(* IEC 61131-3 sources: codesys-mcp-toolkit/standalone-sync/sources_st/511_05/Util, 8 files *)

(* ---- E_InfluxType.dut.st ---- *)
// @OBJECT_ID: 731e7745-b82f-47eb-ba89-92034cdd1c59
// @DECLARATION
TYPE E_InfluxType :
(
    REAL_TYPE,
    INT_TYPE,
    BOOL_TYPE
);
END_TYPE

(* ---- E_InfluxType_1.dut.st ---- *)
// @OBJECT_ID: 96c42348-4289-44bb-9086-91ce752858fa
// @DECLARATION
TYPE E_InfluxType_1 :
(
    REAL_TYPE,
    INT_TYPE,
    BOOL_TYPE
);
END_TYPE

(* ---- U_WordToReal.dut.st ---- *)
// @OBJECT_ID: 3d2ce4b8-1645-47ac-8a08-67d49366f794
// @DECLARATION
TYPE U_WordToReal :
UNION
    dwValue : DWORD; // Используется для битовых операций
    rValue  : REAL;  // Используется для получения результата
END_UNION
END_TYPE

(* ---- AIToFloat.func.st ---- *)
// @OBJECT_ID: 807a566b-cc68-4261-8820-1605cd0b0d30
// @DECLARATION
	FUNCTION AIToFloat : REAL
VAR_INPUT
	In:UINT;
	Lo,Hi:REAL;
END_VAR
VAR
END_VAR

// @IMPLEMENTATION
AIToFloat:=(UINT_TO_REAL(In)-10000.0)/40000.0*Hi+Lo;
//AIToFloat:=(UINT_TO_REAL(In)-0.0)/50000.0*Hi+Lo;

(* ---- FC_ModbusToRealSwapped.func.st ---- *)
// @OBJECT_ID: 0315c496-40b5-48b0-ae72-f392c63e890a
// @DECLARATION
FUNCTION FC_ModbusToRealSwapped : REAL
VAR_INPUT
    wWord1   : WORD;   (* Первое слово из Modbus (например, 53126) *)
    wWord2   : WORD;   (* Второе слово из Modbus (например, 0) *)
END_VAR
VAR
    dwTarget : DWORD;  (* Буфер для сборки 32-битного значения *)
    wTemp1   : WORD;   (* Временные переменные для перестановки байт *)
    wTemp2   : WORD;
    pReal    : POINTER TO REAL; (* Указатель для копирования памяти *)
END_VAR

// @IMPLEMENTATION

(* 1. Переставляем байты внутри каждого слова *)
wTemp1 := ROR(wWord1, 8); (* 0xED0C станет 0x0CED *)
wTemp2 := ROR(wWord2, 8); (* 0x0000 останется 0x0000 *)

(* 2. Собираем DWORD в режиме Little-Endian (wTemp2 сдвигаем в старшие биты) *)
dwTarget := SHL(WORD_TO_DWORD(wTemp2), 16) OR WORD_TO_DWORD(wTemp1);
(* На выходе соберется строка 0x41CD0000 *)

(* 3. Копируем область памяти в REAL *)
pReal := ADR(dwTarget);
FC_ModbusToRealSwapped := pReal^;

(* ---- FloatToAI.func.st ---- *)
// @OBJECT_ID: 9798738f-911b-4eef-bb17-69dfaa9c6f1e
// @DECLARATION
FUNCTION FloatToAI : UINT
VAR_INPUT
	In:REAL;

END_VAR
VAR
END_VAR

// @IMPLEMENTATION
FloatToAI:=REAL_TO_UINT(In/100.0*40000.0+10000.0);

(* ---- Check_Block.fb.st ---- *)
// @OBJECT_ID: a53145cf-05f5-44e2-98c8-5640a1ec8c65
// @DECLARATION
FUNCTION_BLOCK Check_Block
VAR_INPUT
	State_Mixer : BOOL;
	Weight : REAL;
END_VAR
VAR_OUTPUT
	State_Block : BOOL;
	State_Block_P102 : BOOL;
END_VAR
VAR
END_VAR

// @IMPLEMENTATION
IF NOT State_Mixer THEN
	State_Block := TRUE;
ELSE
	State_Block := FALSE;
END_IF;
IF Weight > 3000 THEN
	State_Block_P102 := TRUE;
ELSE
	State_Block_P102 := FALSE;
END_IF;

(* ---- FB_InfluxUdpSender.fb.st ---- *)
// @OBJECT_ID: e559a9a1-9e90-4a38-bf45-4143c502a1fc
// @DECLARATION
FUNCTION_BLOCK FB_InfluxUdpSender
VAR_INPUT
	sSendData : STRING(2000); // Data to send
    sIPInflux : STRING :='192.168.215.5'; // InfluxIP
    uiPortInflux : UINT := 8089; // Influx port
END_VAR
VAR
	eState: 			CLIENT_STATE;								// Шаг состояния клиента

	fbUdpPeer: 			NBS.UDP_Peer;								// ФБ создания UDP-пира
	fbUdpSend: 			NBS.UDP_Send;								// ФБ отправки данных
	sendData : STRING(2000); // Data to send
    numberOfBytesToSend : UDINT := 0; // Number of bytes to send
	influxIP: NBS.IP_ADDR;

	fbSendTrig:			R_TRIG;										// Триггер записи

	blinker:BLINK;
	TimeCycle: TIME:= T#10S;
	bStart : BOOL := FALSE;
END_VAR

// @IMPLEMENTATION
	blinker(ENABLE:=bStart,timelow:=TimeCycle, timehigh:=T#1S);

CASE eState OF

	CLIENT_STATE.CREATE:	// создаем UDP-пира на заданном порту

		fbUdpPeer
		(
			xEnable		:= TRUE,
			ipAddr		:= ,
			uiPort		:= ,
			ipMultiCast	:= ,
		);

		IF fbUdpPeer.xActive THEN
			bStart := TRUE;
			eState	:= CLIENT_STATE.WAITING;
			influxIP.sAddr:=sIPInflux;
		ELSIF fbUdpPeer.xError THEN
			; // обработка ошибок
		END_IF

	CLIENT_STATE.WAITING:	// ожидаем команды на запись

		fbSendTrig(CLK:=blinker.OUT);

		IF fbSendTrig.Q THEN
// Calculate number of bytes to send
			sendData := sSendData;
			numberOfBytesToSend := DINT_TO_UDINT(Stu.StrLenA(ADR(sendData)));

			eState	:= CLIENT_STATE.SEND;
		END_IF

	CLIENT_STATE.SEND:		// отправляем запрос серверу

			fbUdpSend
			(
				xExecute	:=	TRUE,
				udiTimeOut:= 1000,
				hPeer		:=	fbUdpPeer.hPeer,
				ipAddr:=  influxIP,
				uiPort:= uiPortInflux,
				szSize:= numberOfBytesToSend,
				pData:= ADR(sendData),
			);

			IF (fbUdpSend.xDone OR fbUdpSend.xError) THEN
				fbUdpSend(xExecute:=FALSE);
				eState	:= 	CLIENT_STATE.WAITING;
			END_IF

END_CASE
